// TIA Portal project "car_turn_signal" (V16)

(* hardware
DEVICE "S7-1200 station_1"  S7-1200 Station
   slot 0: "Rack_0"  S7-1200 Rack  Rack  V1.0
   slot 1: "PLC_1"  CPU 1212C DC/DC/DC  6ES7 212-1AE40-0XB0  V4.4
DEVICE "HMI_1"  TP700 Comfort
   slot 0: "HMI_1"  TP700 Comfort  6AV2 124-0GC01-0AX0  16.0.0.0
   slot 1: "HMI_RT_1"  TP700 Comfort  6AV2 124-0GC01-0AX0  16.0.0.0
   slot 5: "HMI_1.IE_CP_1"  PROFINET Interface  16.0.0.0
      slot 1: "PROFINET Interface_1"  PROFINET Interface
         slot 1: "Port_1"  Port
         slot 2: "Port_2"  Port
   slot 7: "HMI_1.MPI/DP_CP_1"  MPI/DP Interface  16.0.0.0
*)

// ===== PLC "PLC_1"  CPU 1212C DC/DC/DC =====

VAR_GLOBAL   // PLC tag table "默认变量表"
   "left" AT %M3.0 : Bool;
   "Right" AT %M3.1 : Bool;
   "OutLeft" AT %Q0.0 : Bool;
   "OutRight" AT %Q0.1 : Bool;
   "System_Byte" AT %MB1 : Byte;
   "FirstScan" AT %M1.0 : Bool;
   "DiagStatusUpdate" AT %M1.1 : Bool;
   "AlwaysTRUE" AT %M1.2 : Bool;
   "AlwaysFALSE" AT %M1.3 : Bool;
   "Clock_Byte" AT %MB0 : Byte;
   "Clock_10Hz" AT %M0.0 : Bool;
   "Clock_5Hz" AT %M0.1 : Bool;
   "Clock_2.5Hz" AT %M0.2 : Bool;
   "Clock_2Hz" AT %M0.3 : Bool;
   "Clock_1.25Hz" AT %M0.4 : Bool;
   "Clock_1Hz" AT %M0.5 : Bool;
   "Clock_0.625Hz" AT %M0.6 : Bool;
   "Clock_0.5Hz" AT %M0.7 : Bool;
   "Tag_1" AT %M2.1 : Bool;
   "Tag_2" AT %M2.0 : Bool;
   "Reset" AT %M3.2 : Bool;
END_VAR

// folder: System blocks/Program resources

DATA_BLOCK "IEC_Timer_0_DB_1"   // DB2
{ S7_Optimized_Access := 'TRUE' }
AUTHOR : Simatic
FAMILY : IEC
NAME : IEC_TMR
VERSION : 1.0
// stored: InstanceOfName IEC_TIMER
"IEC_TIMER"
BEGIN
END_DATA_BLOCK

// folder: (top level)

ORGANIZATION_BLOCK "Main"   // OB1, LAD, ProgramCycle
TITLE = "Main Program Sweep (Cycle)"
{ S7_Optimized_Access := 'TRUE' }
VERSION : 0.1
   VAR_INPUT
      Initial_Call : Bool;   // Initial call of this OB
      Remanence : Bool;   // =True, if remanent data are available
   END_VAR
   VAR_TEMP   // added for the SCL form of the ladder/FBD networks
      _w1 : Bool;
   END_VAR
BEGIN

REGION Network 1
   // left
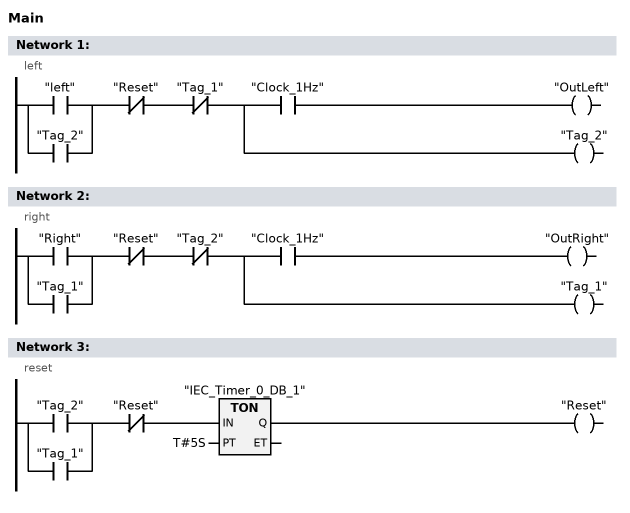
   RUNG wire#powerrail
      Contact( "left" )
      wire#w1
      I_Contact( "Reset" )
      I_Contact( "Tag_1" )
      wire#w2
      Contact( "Clock_1Hz" )
      Coil( "OutLeft" )
   END_RUNG
   RUNG wire#powerrail
      Contact( "Tag_2" )
   END_RUNG wire#w1
   RUNG wire#w2
      Coil( "Tag_2" )
   END_RUNG
   // the same network as SCL:
   #_w1 := ("left" OR "Tag_2") AND NOT "Reset" AND NOT "Tag_1";
   "OutLeft" := #_w1 AND "Clock_1Hz";
   "Tag_2" := #_w1;
END_REGION

REGION Network 2
   // right
   RUNG wire#powerrail
      Contact( "Right" )
      wire#w1
      I_Contact( "Reset" )
      I_Contact( "Tag_2" )
      wire#w2
      Contact( "Clock_1Hz" )
      Coil( "OutRight" )
   END_RUNG
   RUNG wire#powerrail
      Contact( "Tag_1" )
   END_RUNG wire#w1
   RUNG wire#w2
      Coil( "Tag_1" )
   END_RUNG
   // the same network as SCL:
   #_w1 := ("Right" OR "Tag_1") AND NOT "Reset" AND NOT "Tag_2";
   "OutRight" := #_w1 AND "Clock_1Hz";
   "Tag_1" := #_w1;
END_REGION

REGION Network 3
   // reset
   "IEC_Timer_0_DB_1".TON(IN := ("Tag_2" OR "Tag_1") AND NOT "Reset", PT := T#5S);
   "Reset" := "IEC_Timer_0_DB_1".Q;
END_REGION
END_ORGANIZATION_BLOCK

(* ===== HMI "HMI_RT_1" =====
system functions are stored by id; their names below are inferred from use
connection "HMI_连接_1": ETHERNET, S7_1200_OMS

HMI tags "默认变量表"
   "left" : Bool = PLC left AT %M3.0, 1 s
   "Reset" : Bool = PLC Reset AT %M3.2, 1 s
   "Right" : Bool = PLC Right AT %M3.1, 1 s
   "OutLeft" : Bool = PLC OutLeft AT %Q0.0, 1 s
   "OutRight" : Bool = PLC OutRight AT %Q0.1, 1 s

screen "画面_1" 800x480
   Button "按钮_1" at 189,272 size 106x61; TextOff 'Left'
      on Press: SetBit("left")
      on Release: ResetBit("left")
   Button "按钮_2" at 492,272 size 106x61; TextOff 'Right'
      on Press: SetBit("Right")
      on Release: ResetBit("Right")
   Polygon "多边形_1" at 251,92 size 74x85
      Appearance <- "OutLeft"
   Polygon "多边形_2" at 440,92 size 71x85
      Appearance <- "OutRight"
   Button "按钮_3" at 337,272 size 106x61; TextOff 'Reset'
      on Press: SetBit("Reset")
      on Release: ResetBit("Reset")
*)